PROGRAM FAST
VAR
	instFB_MetricsAndCalculation: FB_MetricsAndCalculation;
	
END_VAR

_00_UpdateHardware();
_03_MetricsAndCalculation();

(*==============================================================================================================================
CPNTeck - Automação industrial
(c)Copyright 2023 All Rights Reserved
_______________________________________________________________________________________________________________________________
Library: <N/A or library name>
Tested with: <PLC / IPC model>
Engineering: <TwinCAT version>
Restrictions: <text>
Requirements: <text>
Functionality: <short description>
Support: <email>
Note: Parameter comments are only available in language 'English (United States)'
_______________________________________________________________________________________________________________________________
Change log table:

Version  		| Date        			| Expert in charge  	| Changes applied
<xx.xx.xx>		| <dd.mm.yyyy>  		| <name>              | <changes>

===============================================================================================================================*)

METHOD _00_UpdateHardware
VAR_INPUT
END_VAR
SLT1_P1_050_DI01();
SLT1_P1_050_DI02();
SLT1_P1_050_DI03();
SLT1_P1_050_DI04();
SLT1_P1_050_DI05();
SLT1_P1_050_DI06();

SLT1_P1_050_DO01();
SLT1_P1_050_DO02();
SLT1_P1_050_DO03();
SLT1_P1_050_DO04();
SLT1_P1_050_DO05();
SLT1_P1_050_DO06();

ARK_P1_050_DI01();
ARK_P1_050_DO01();
ARK_P1_050_DO02();

ARK_P1_050_AI01();
ARK_P1_050_AO01();	
ARK_P1_050_AO02();
END_METHOD

METHOD _03_MetricsAndCalculation
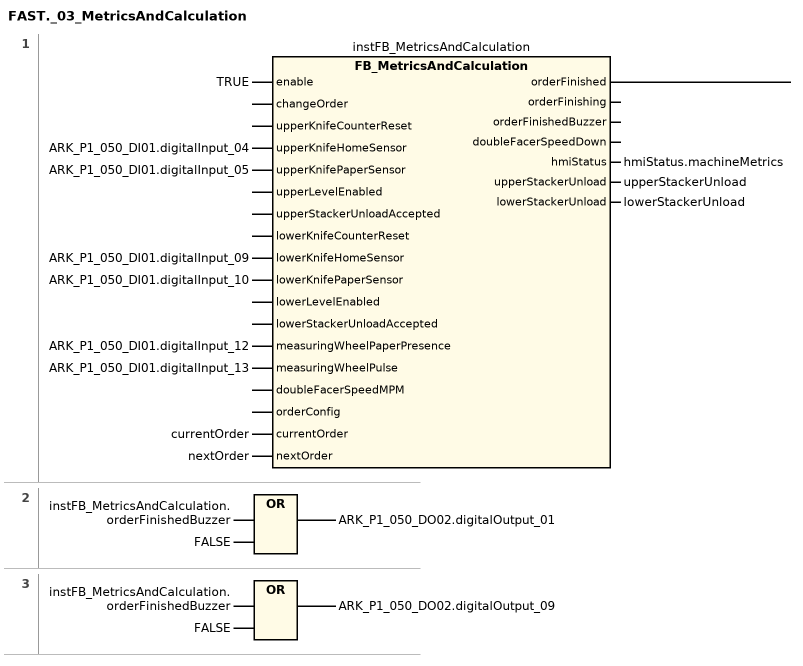
// NETWORK 1
instFB_MetricsAndCalculation(
    enable := TRUE,
    upperKnifeHomeSensor := ARK_P1_050_DI01.digitalInput_04,
    upperKnifePaperSensor := ARK_P1_050_DI01.digitalInput_05,
    lowerKnifeHomeSensor := ARK_P1_050_DI01.digitalInput_09,
    lowerKnifePaperSensor := ARK_P1_050_DI01.digitalInput_10,
    measuringWheelPaperPresence := ARK_P1_050_DI01.digitalInput_12,
    measuringWheelPulse := ARK_P1_050_DI01.digitalInput_13,
    currentOrder := currentOrder,
    nextOrder := nextOrder,
    hmiStatus => hmiStatus.machineMetrics,
    upperStackerUnload => upperStackerUnload,
    lowerStackerUnload => lowerStackerUnload); // FB_MetricsAndCalculation

// NETWORK 2
ARK_P1_050_DO02.digitalOutput_01 := instFB_MetricsAndCalculation.orderFinishedBuzzer OR FALSE;

// NETWORK 3
ARK_P1_050_DO02.digitalOutput_09 := instFB_MetricsAndCalculation.orderFinishedBuzzer OR FALSE;
END_METHOD

END_PROGRAM

(* stored: Version 1.1.0.1
   POU FAST: Id {9d8a0c7e-5072-4f3b-9af3-b5e9562092cd}, SpecialFunc None
   Method _00_UpdateHardware: Id {d837d4b8-5249-4ca0-8b29-9b01e83b86fc}
   Method _03_MetricsAndCalculation: Id {9f336ba8-4427-4aa8-a37a-86092c6673e6} *)
